(* LS Electric XG5000 project: XEM_SS2_ModRTU_Example *)
(* PLC LSPLC *)
(* module base 0 slot 0: Input/Output Module:XEM-DN/DP32HP (DC 24V Input, Transistor Output, 32 Contacts) *)
(* module base 0 slot 1: Internal Positioning:XBF-PO06E (Open Collector Type, 6 Axis) *)
VAR_GLOBAL
    gRead_Mapping_Registers AT %MW10 : ARRAY[0..3] OF WORD; (* Mapping Registers buffer configured for Read Only.  There are 2 parameters that are 2 words of data each *)
    gStatus_Monitor_Registers AT %MW0 : ARRAY[0..9] OF WORD; (* Status Monitor register buffer.  There are 5 parameters that are 2 words of data each. *)
    gWrite_Mapping_Registers AT %MW14 : ARRAY[0..7] OF WORD; (* Mapping registers buffer configured for writing data. There are 4 parameters that are 2 words of data each *)
    SS2_Drive00 : SureServo2_UDT; (* SS2 data type for drive 00 *)
END_VAR

TYPE SureServo2_UDT : (* Data type for accessing inputs and outputs of a SureServo2. *)
STRUCT
    Status_Z_Phase_Offset : DINT; (* z phase offset of Sure servo 2 *)
    Status_Position_Feedback : DINT; (* current position *)
    Status_Speed_Feedback : DINT; (* current speed *)
    Status_Torque_Feedback : DINT; (* current torque *)
    Integrated_DI_Status : DWORD; (* integrated digital inputs *)
    Status_Servo_Alarm : INT; (* current servo alarm *)
    Status_Path_Target_Status : INT; (* status of path target command.  servo should be in PR control mode. *)
    Status_Servo_Ready : BOOL; (* Servo is ready for commands *)
    Status_Servo_Enabled : BOOL; (* Servo has been enabled *)
    Status_Zero_Speed : BOOL; (* Servo is at zero speed *)
    Status_Target_Speed_Reached : BOOL; (* target speed has been reached *)
    Status_Target_Position_Reached : BOOL; (* target position has been reached *)
    Status_Torque_Limit_Reached : BOOL; (* torque limit has been reached. *)
    Status_Alarm : BOOL; (* drive alarm status *)
    Status_Brake_On : BOOL; (* motor brake status *)
    Status_Home : BOOL; (* axis is at home. *)
    Status_Motor_Overload : BOOL; (* status that the motor is overloaded *)
    Status_Warning : BOOL; (* status that there is a drive warning. *)
    Control_Speed_CMD3 : DINT; (* speed command *)
    Control_Servo_Enable : BOOL; (* command to enable the servo *)
    Control_Alarm_Reset : BOOL; (* command to reset an alarm *)
    Control_Speed_PR_Mode : BOOL; (* command for speed or path target mode *)
    Control_Trigger : BOOL; (* trigger command *)
    Control_PR_Select_0 : BOOL; (* path target mode 0 *)
    Control_Stop : BOOL; (* Stop motion command *)
    Control_EStop : BOOL; (* emergency stop status *)
    Control_ECAM_On : BOOL; (* command to turn on ECAM functionality *)
    Control_PR_Path_Target : UINT; (* Path target value *)
    Control_PR_Path_Trigger : UINT; (* Path target trigger value. *)
END_STRUCT;
END_TYPE

PROGRAM Drive_Control_Program (* task: Scan Program *)
VAR_EXTERNAL
    gStatus_Monitor_Registers : ARRAY[0..9] OF WORD; (* AT %MW0 *) (* Status Monitor register buffer.  There are 5 parameters that are 2 words of data each. *)
    gWrite_Mapping_Registers : ARRAY[0..7] OF WORD; (* AT %MW14 *) (* Mapping registers buffer configured for writing data. There are 4 parameters that are 2 words of data each *)
    SS2_Drive00 : SureServo2_UDT; (* SS2 data type for drive 00 *)
END_VAR
VAR
    tempDword : DWORD; (* temporary DWORD storage for *)
END_VAR

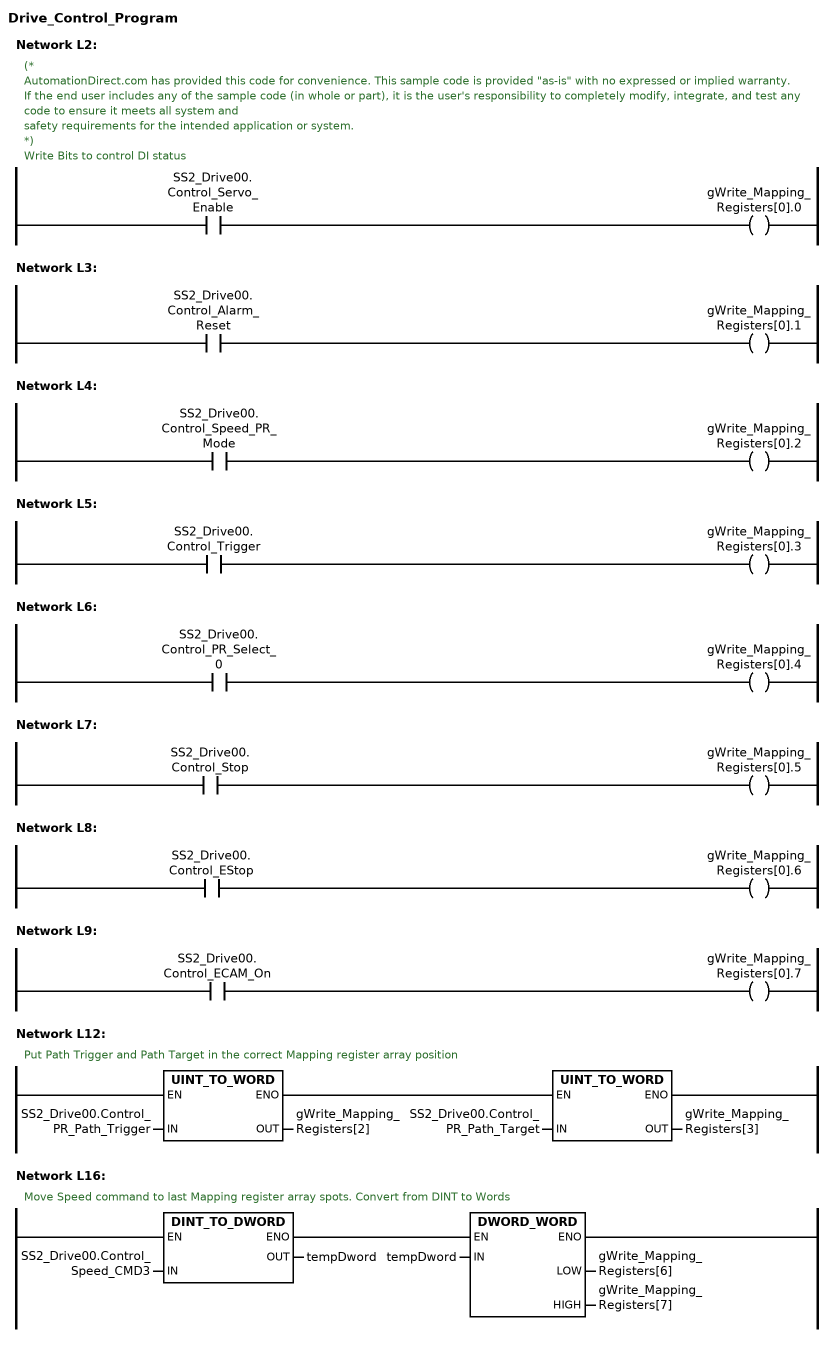
(* ( * / AutomationDirect.com has provided this code for convenience. This sample code is provided "as-is" with no expressed or implied warranty. / If the end user includes any of the sample code (in whole or part), it is the user's responsibility to completely modify, integrate, and test any code to ensure it meets all system and / safety requirements for the intended application or system. / * ) *)
(* Write Bits to control DI status *)
(* Rung L2 *)
gWrite_Mapping_Registers[0].0 := SS2_Drive00.Control_Servo_Enable;
(* Rung L3 *)
gWrite_Mapping_Registers[0].1 := SS2_Drive00.Control_Alarm_Reset;
(* Rung L4 *)
gWrite_Mapping_Registers[0].2 := SS2_Drive00.Control_Speed_PR_Mode;
(* Rung L5 *)
gWrite_Mapping_Registers[0].3 := SS2_Drive00.Control_Trigger;
(* Rung L6 *)
gWrite_Mapping_Registers[0].4 := SS2_Drive00.Control_PR_Select_0;
(* Rung L7 *)
gWrite_Mapping_Registers[0].5 := SS2_Drive00.Control_Stop;
(* Rung L8 *)
gWrite_Mapping_Registers[0].6 := SS2_Drive00.Control_EStop;
(* Rung L9 *)
gWrite_Mapping_Registers[0].7 := SS2_Drive00.Control_ECAM_On;
(* Put Path Trigger and Path Target in the correct Mapping register array position *)
(* Rung L12 *)
gWrite_Mapping_Registers[2] := UINT_TO_WORD(SS2_Drive00.Control_PR_Path_Trigger);
gWrite_Mapping_Registers[3] := UINT_TO_WORD(SS2_Drive00.Control_PR_Path_Target);
(* Move Speed command to last Mapping register array spots. Convert from DINT to Words *)
(* Rung L16 *)
tempDword := DINT_TO_DWORD(SS2_Drive00.Control_Speed_CMD3);
gWrite_Mapping_Registers[6] := DWORD_WORD(IN := tempDword, HIGH => gWrite_Mapping_Registers[7]);
END_PROGRAM

PROGRAM Drive_Status_Program (* task: Scan Program *)
VAR_EXTERNAL
    gRead_Mapping_Registers : ARRAY[0..3] OF WORD; (* AT %MW10 *) (* Mapping Registers buffer configured for Read Only.  There are 2 parameters that are 2 words of data each *)
    gStatus_Monitor_Registers : ARRAY[0..9] OF WORD; (* AT %MW0 *) (* Status Monitor register buffer.  There are 5 parameters that are 2 words of data each. *)
    SS2_Drive00 : SureServo2_UDT; (* SS2 data type for drive 00 *)
END_VAR
VAR
    tempDword : DWORD; (* temporary DWORD storage for *)
END_VAR

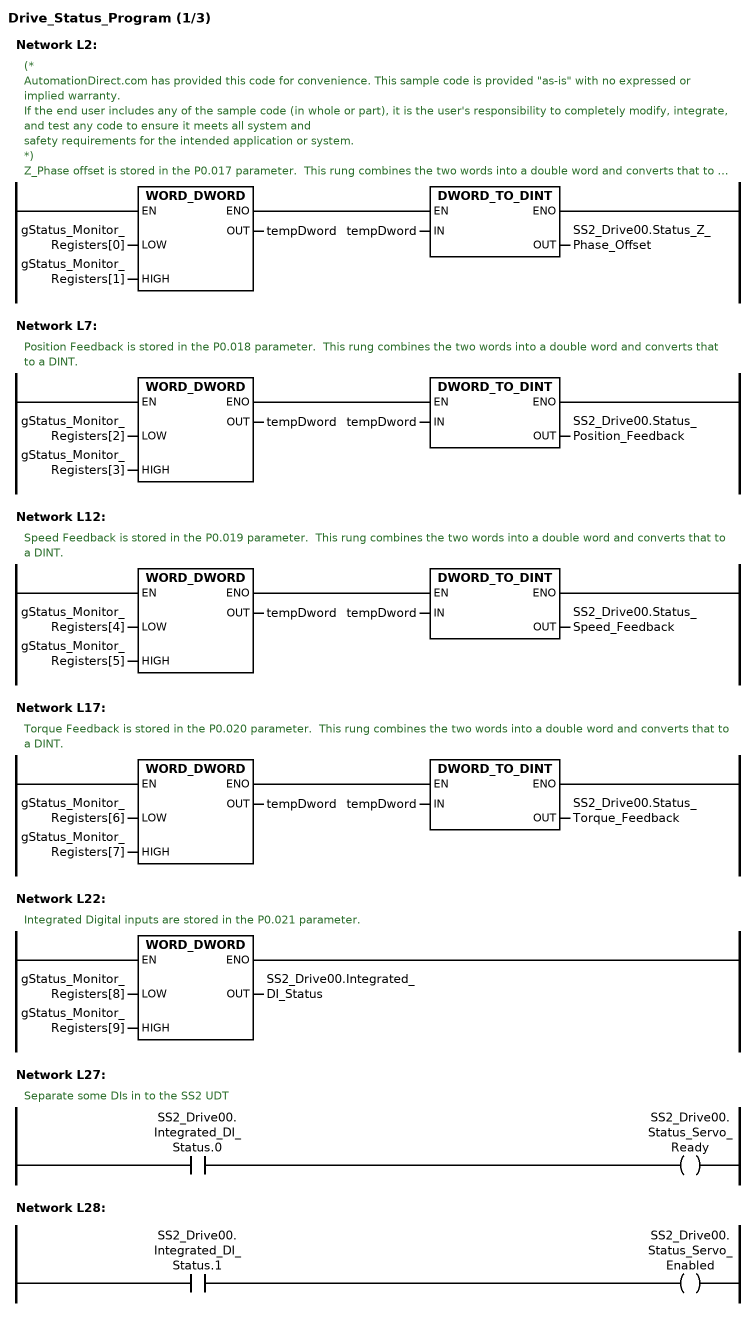
(* ( * / AutomationDirect.com has provided this code for convenience. This sample code is provided "as-is" with no expressed or implied warranty. / If the end user includes any of the sample code (in whole or part), it is the user's responsibility to completely modify, integrate, and test any code to ensure it meets all system and / safety requirements for the intended application or system. / * ) *)
(* Z_Phase offset is stored in the P0.017 parameter.  This rung combines the two words into a double word and converts that to a DINT. *)
(* Rung L2 *)
tempDword := WORD_DWORD(LOW := gStatus_Monitor_Registers[0], HIGH := gStatus_Monitor_Registers[1]);
SS2_Drive00.Status_Z_Phase_Offset := DWORD_TO_DINT(tempDword);
(* Position Feedback is stored in the P0.018 parameter.  This rung combines the two words into a double word and converts that to a DINT. *)
(* Rung L7 *)
tempDword := WORD_DWORD(LOW := gStatus_Monitor_Registers[2], HIGH := gStatus_Monitor_Registers[3]);
SS2_Drive00.Status_Position_Feedback := DWORD_TO_DINT(tempDword);
(* Speed Feedback is stored in the P0.019 parameter.  This rung combines the two words into a double word and converts that to a DINT. *)
(* Rung L12 *)
tempDword := WORD_DWORD(LOW := gStatus_Monitor_Registers[4], HIGH := gStatus_Monitor_Registers[5]);
SS2_Drive00.Status_Speed_Feedback := DWORD_TO_DINT(tempDword);
(* Torque Feedback is stored in the P0.020 parameter.  This rung combines the two words into a double word and converts that to a DINT. *)
(* Rung L17 *)
tempDword := WORD_DWORD(LOW := gStatus_Monitor_Registers[6], HIGH := gStatus_Monitor_Registers[7]);
SS2_Drive00.Status_Torque_Feedback := DWORD_TO_DINT(tempDword);
(* Integrated Digital inputs are stored in the P0.021 parameter. *)
(* Rung L22 *)
SS2_Drive00.Integrated_DI_Status := WORD_DWORD(LOW := gStatus_Monitor_Registers[8], HIGH := gStatus_Monitor_Registers[9]);
(* Separate some DIs in to the SS2 UDT *)
(* Rung L27 *)
SS2_Drive00.Status_Servo_Ready := SS2_Drive00.Integrated_DI_Status.0;
(* Rung L28 *)
SS2_Drive00.Status_Servo_Enabled := SS2_Drive00.Integrated_DI_Status.1;

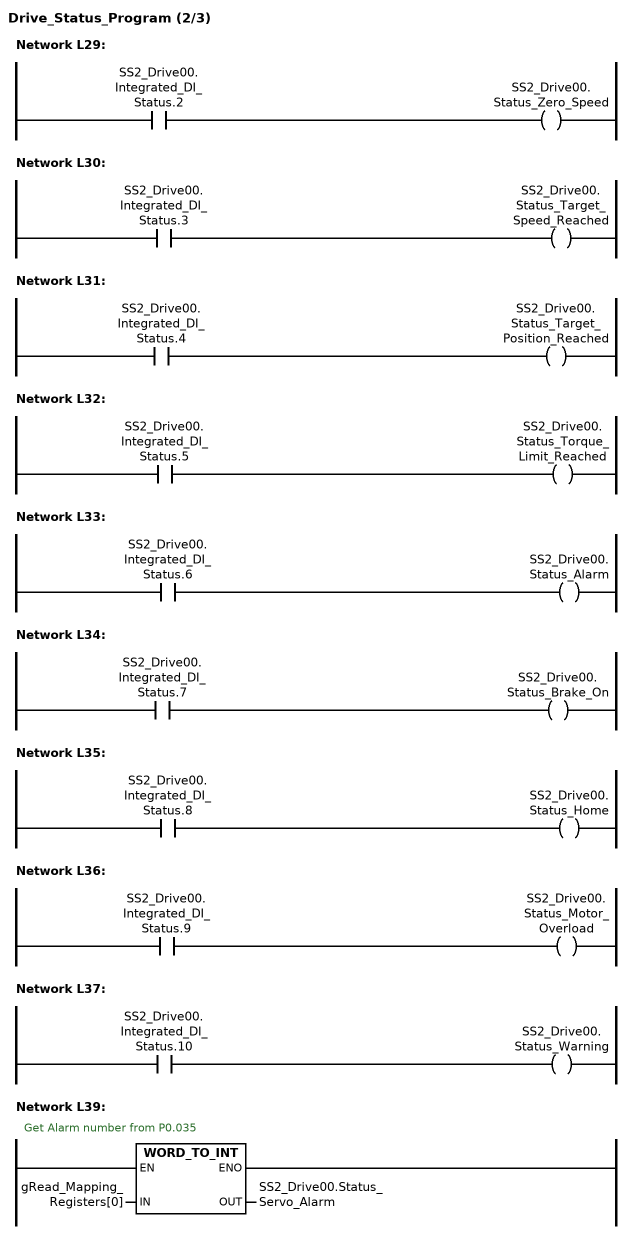
(* Rung L29 *)
SS2_Drive00.Status_Zero_Speed := SS2_Drive00.Integrated_DI_Status.2;
(* Rung L30 *)
SS2_Drive00.Status_Target_Speed_Reached := SS2_Drive00.Integrated_DI_Status.3;
(* Rung L31 *)
SS2_Drive00.Status_Target_Position_Reached := SS2_Drive00.Integrated_DI_Status.4;
(* Rung L32 *)
SS2_Drive00.Status_Torque_Limit_Reached := SS2_Drive00.Integrated_DI_Status.5;
(* Rung L33 *)
SS2_Drive00.Status_Alarm := SS2_Drive00.Integrated_DI_Status.6;
(* Rung L34 *)
SS2_Drive00.Status_Brake_On := SS2_Drive00.Integrated_DI_Status.7;
(* Rung L35 *)
SS2_Drive00.Status_Home := SS2_Drive00.Integrated_DI_Status.8;
(* Rung L36 *)
SS2_Drive00.Status_Motor_Overload := SS2_Drive00.Integrated_DI_Status.9;
(* Rung L37 *)
SS2_Drive00.Status_Warning := SS2_Drive00.Integrated_DI_Status.10;
(* Get Alarm number from P0.035 *)
(* Rung L39 *)
SS2_Drive00.Status_Servo_Alarm := WORD_TO_INT(gRead_Mapping_Registers[0]);

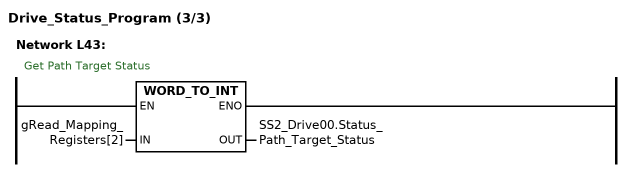
(* Get Path Target Status *)
(* Rung L43 *)
SS2_Drive00.Status_Path_Target_Status := WORD_TO_INT(gRead_Mapping_Registers[2]);
END_PROGRAM